// TIA Portal V15.1 export
// export: Created 2024-06-21T08:40:52.289879Z, ExportSetting WithDefaults, DisplayName Totally Integrated Automation Portal, DisplayVersion V15.1 Update 5, DisplayName TIA Portal Openness, DisplayVersion V15.1 Update 5, DisplayName SINAMICS Startdrive Advanced, DisplayVersion V15.1, DisplayName G130, G150, S120, S150, SINAMICS MV, S210, DisplayVersion V15.1, DisplayName G110M, G120, G120C, G120D, G120P, DisplayVersion V15.1, DisplayName STEP 7 Professional, DisplayVersion V15.1 Update 5, DisplayName STEP 7 Safety, DisplayVersion V15.1, DisplayName WinCC Professional, DisplayVersion V15.1 Update 5, DisplayName SIMATIC Visualization Architect, DisplayVersion V15.1
FUNCTION "F209230ZS01Input" : Void   // FC7030, F_FBD
TITLE = Safety Inputs ZMProc / Safety Inputs 209230ZS01
{ S7_Optimized_Access := 'TRUE' }
VERSION : 0.1
// stored: AutoNumber false, IsIECCheckEnabled false, UDAEnableTagReadback false
BEGIN

REGION Network 1: **** 1 - Inputs **** 209230AS10 Reset command Input
   // Reset command Input
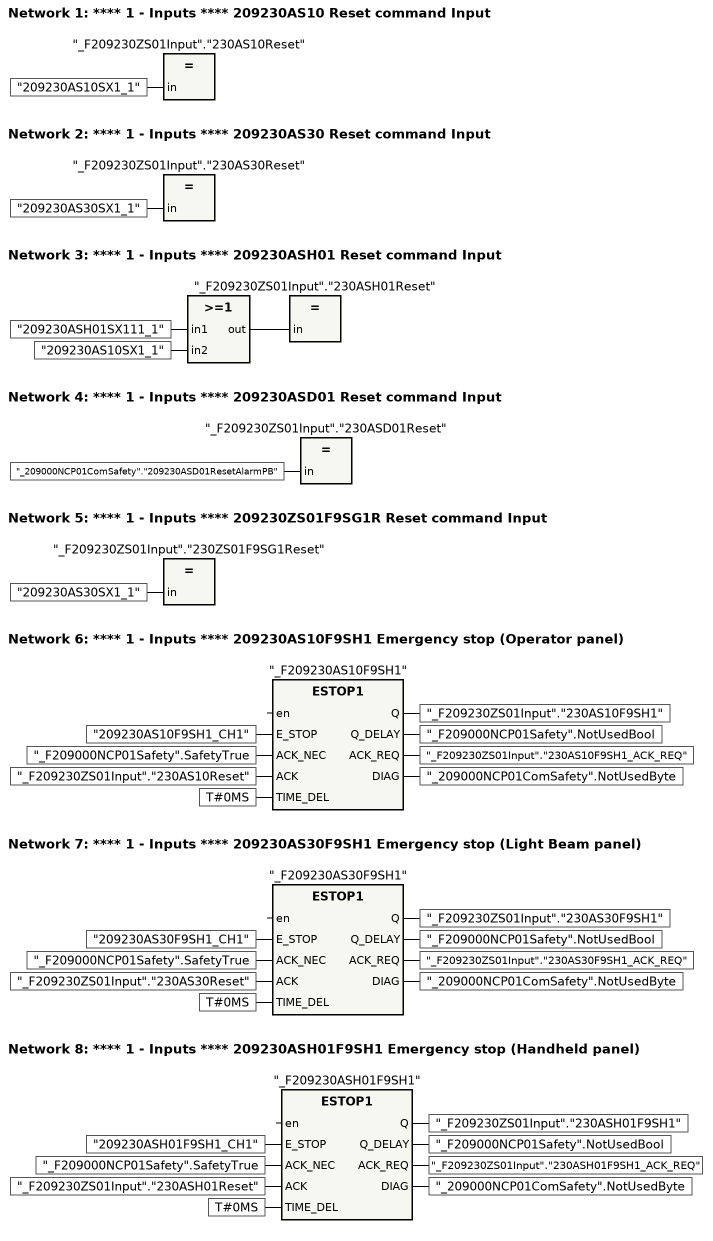
   "_F209230ZS01Input"."230AS10Reset" := "209230AS10SX1_1";
END_REGION

REGION Network 2: **** 1 - Inputs **** 209230AS30 Reset command Input
   // Reset command Input
   "_F209230ZS01Input"."230AS30Reset" := "209230AS30SX1_1";
END_REGION

REGION Network 3: **** 1 - Inputs **** 209230ASH01 Reset command Input
   // Reset command Input
   "_F209230ZS01Input"."230ASH01Reset" := "209230ASH01SX111_1" OR "209230AS10SX1_1";
END_REGION

REGION Network 4: **** 1 - Inputs **** 209230ASD01 Reset command Input
   // Reset command Input
   "_F209230ZS01Input"."230ASD01Reset" := "_209000NCP01ComSafety"."209230ASD01ResetAlarmPB";
END_REGION

REGION Network 5: **** 1 - Inputs **** 209230ZS01F9SG1R Reset command Input
   // Reset command Input
   "_F209230ZS01Input"."230ZS01F9SG1Reset" := "209230AS30SX1_1";
END_REGION

REGION Network 6: **** 1 - Inputs **** 209230AS10F9SH1 Emergency stop (Operator panel)
   // Emergency Stop
   "_F209230AS10F9SH1"(E_STOP := "209230AS10F9SH1_CH1",   // ESTOP1
                       ACK_NEC := "_F209000NCP01Safety".SafetyTrue,
                       ACK := "_F209230ZS01Input"."230AS10Reset",
                       TIME_DEL := T#0MS,
                       Q => "_F209230ZS01Input"."230AS10F9SH1",
                       Q_DELAY => "_F209000NCP01Safety".NotUsedBool,
                       ACK_REQ => "_F209230ZS01Input"."230AS10F9SH1_ACK_REQ",
                       DIAG => "_209000NCP01ComSafety".NotUsedByte);
END_REGION

REGION Network 7: **** 1 - Inputs **** 209230AS30F9SH1 Emergency stop (Light Beam panel)
   // Emergency Stop
   "_F209230AS30F9SH1"(E_STOP := "209230AS30F9SH1_CH1",   // ESTOP1
                       ACK_NEC := "_F209000NCP01Safety".SafetyTrue,
                       ACK := "_F209230ZS01Input"."230AS30Reset",
                       TIME_DEL := T#0MS,
                       Q => "_F209230ZS01Input"."230AS30F9SH1",
                       Q_DELAY => "_F209000NCP01Safety".NotUsedBool,
                       ACK_REQ => "_F209230ZS01Input"."230AS30F9SH1_ACK_REQ",
                       DIAG => "_209000NCP01ComSafety".NotUsedByte);
END_REGION

REGION Network 8: **** 1 - Inputs **** 209230ASH01F9SH1 Emergency stop (Handheld panel)
   // Emergency Stop
   "_F209230ASH01F9SH1"(E_STOP := "209230ASH01F9SH1_CH1",   // ESTOP1
                        ACK_NEC := "_F209000NCP01Safety".SafetyTrue,
                        ACK := "_F209230ZS01Input"."230ASH01Reset",
                        TIME_DEL := T#0MS,
                        Q => "_F209230ZS01Input"."230ASH01F9SH1",
                        Q_DELAY => "_F209000NCP01Safety".NotUsedBool,
                        ACK_REQ => "_F209230ZS01Input"."230ASH01F9SH1_ACK_REQ",
                        DIAG => "_209000NCP01ComSafety".NotUsedByte);
END_REGION

REGION Network 9: **** 1 - Inputs **** xxxAS05F9SH1 (Emergency Stop) / **** 1 - Inputs **** 209230ASD01F9SH1 Emergency Stop (MGB)
   // Emergency Stop
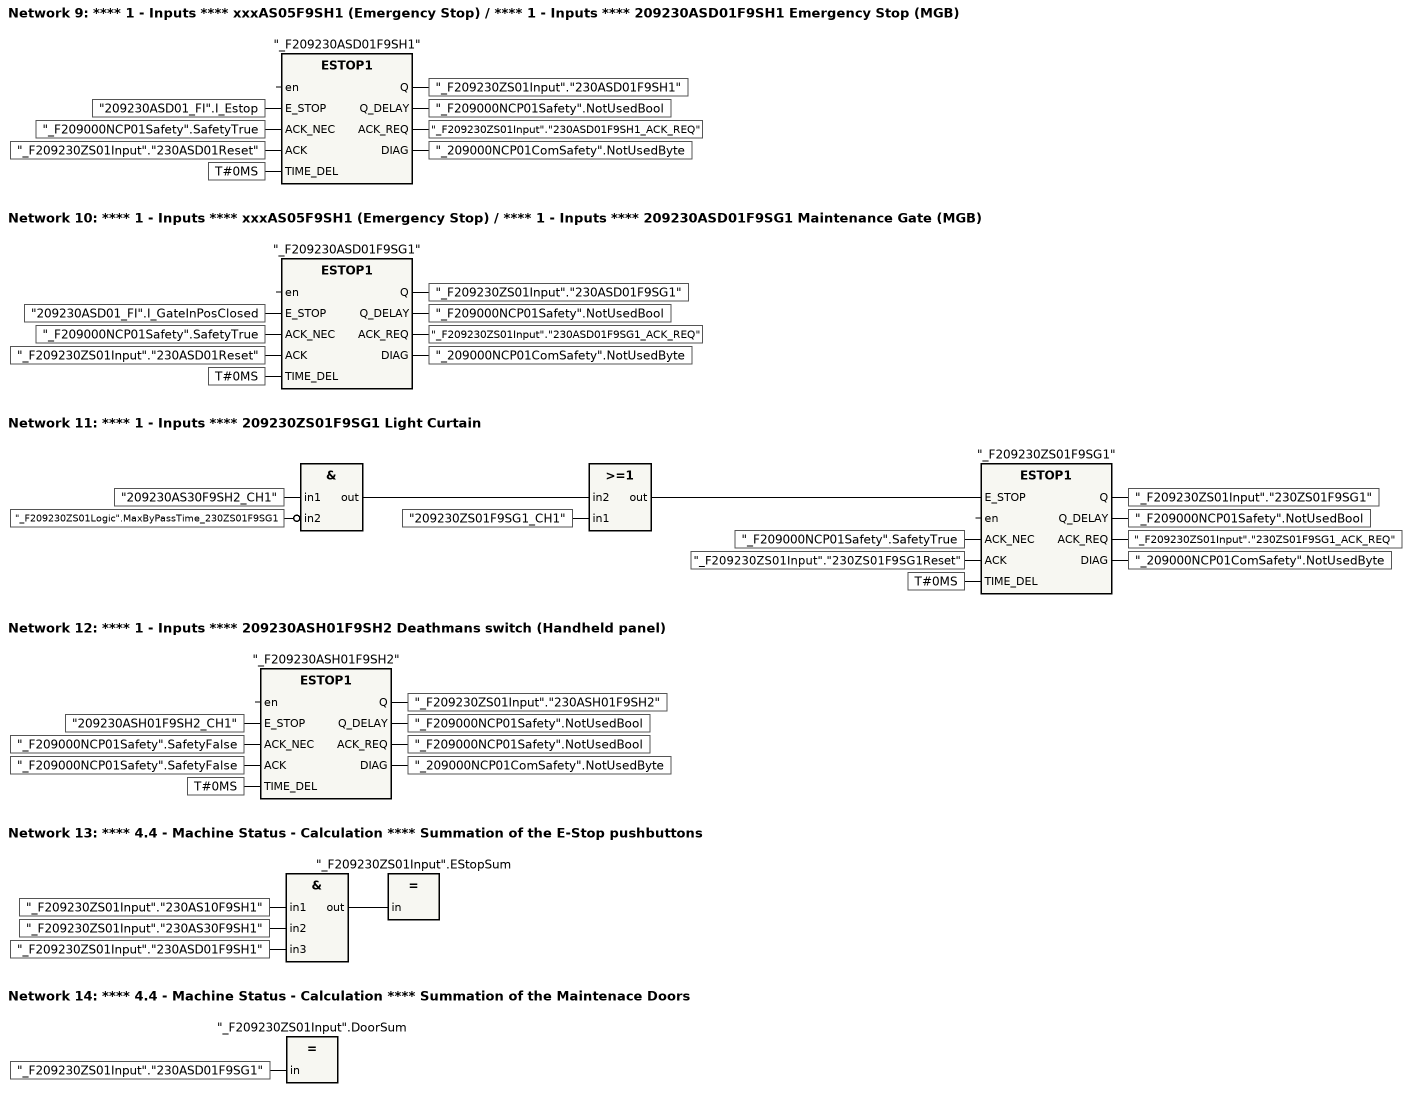
   "_F209230ASD01F9SH1"(E_STOP := "209230ASD01_FI".I_Estop,   // ESTOP1
                        ACK_NEC := "_F209000NCP01Safety".SafetyTrue,
                        ACK := "_F209230ZS01Input"."230ASD01Reset",
                        TIME_DEL := T#0MS,
                        Q => "_F209230ZS01Input"."230ASD01F9SH1",
                        Q_DELAY => "_F209000NCP01Safety".NotUsedBool,
                        ACK_REQ => "_F209230ZS01Input"."230ASD01F9SH1_ACK_REQ",
                        DIAG => "_209000NCP01ComSafety".NotUsedByte);
END_REGION

REGION Network 10: **** 1 - Inputs **** xxxAS05F9SH1 (Emergency Stop) / **** 1 - Inputs **** 209230ASD01F9SG1 Maintenance Gate (MGB)
   // Emergency Stop / Safety Door
   "_F209230ASD01F9SG1"(E_STOP := "209230ASD01_FI".I_GateInPosClosed,   // ESTOP1
                        ACK_NEC := "_F209000NCP01Safety".SafetyTrue,
                        ACK := "_F209230ZS01Input"."230ASD01Reset",
                        TIME_DEL := T#0MS,
                        Q => "_F209230ZS01Input"."230ASD01F9SG1",
                        Q_DELAY => "_F209000NCP01Safety".NotUsedBool,
                        ACK_REQ => "_F209230ZS01Input"."230ASD01F9SG1_ACK_REQ",
                        DIAG => "_209000NCP01ComSafety".NotUsedByte);
END_REGION

REGION Network 11: **** 1 - Inputs **** 209230ZS01F9SG1 Light Curtain
   // Light Curtain
   "_F209230ZS01F9SG1"(E_STOP := ("209230AS30F9SH2_CH1" AND NOT "_F209230ZS01Logic".MaxByPassTime_230ZS01F9SG1) OR "209230ZS01F9SG1_CH1",   // ESTOP1
                       ACK_NEC := "_F209000NCP01Safety".SafetyTrue,
                       ACK := "_F209230ZS01Input"."230ZS01F9SG1Reset",
                       TIME_DEL := T#0MS,
                       Q => "_F209230ZS01Input"."230ZS01F9SG1",
                       Q_DELAY => "_F209000NCP01Safety".NotUsedBool,
                       ACK_REQ => "_F209230ZS01Input"."230ZS01F9SG1_ACK_REQ",
                       DIAG => "_209000NCP01ComSafety".NotUsedByte);
END_REGION

REGION Network 12: **** 1 - Inputs **** 209230ASH01F9SH2 Deathmans switch (Handheld panel)
   // Emergency Stop
   "_F209230ASH01F9SH2"(E_STOP := "209230ASH01F9SH2_CH1",   // ESTOP1
                        ACK_NEC := "_F209000NCP01Safety".SafetyFalse,
                        ACK := "_F209000NCP01Safety".SafetyFalse,
                        TIME_DEL := T#0MS,
                        Q => "_F209230ZS01Input"."230ASH01F9SH2",
                        Q_DELAY => "_F209000NCP01Safety".NotUsedBool,
                        ACK_REQ => "_F209000NCP01Safety".NotUsedBool,
                        DIAG => "_209000NCP01ComSafety".NotUsedByte);
END_REGION

REGION Network 13: **** 4.4 - Machine Status - Calculation **** Summation of the E-Stop pushbuttons
   // Summation of the E-Stop pushbuttons
   "_F209230ZS01Input".EStopSum := "_F209230ZS01Input"."230AS10F9SH1" AND "_F209230ZS01Input"."230AS30F9SH1" AND "_F209230ZS01Input"."230ASD01F9SH1";
END_REGION

REGION Network 14: **** 4.4 - Machine Status - Calculation **** Summation of the Maintenace Doors
   // Summation of the Maintenace Doors
   "_F209230ZS01Input".DoorSum := "_F209230ZS01Input"."230ASD01F9SG1";
END_REGION
END_FUNCTION
